// TIA Portal V19 export
FUNCTION "CollectAlarms" : Void   // FC103, LAD
TITLE = Alarm Collector Unit
// Collects alarms from the respective level and categorises the alarms into the different alarm classes. Filling the alarm DB with specific alarm messages which are defined in the comment of the defined alarm. The definition of possible alarms within a equipment is handled here.
// stored: Namespace Unit2.Em5, SetENOAutomatically false
   VAR_INPUT
      resetAlarms : Bool;
      disableAlarms : Bool;
   END_VAR
   VAR_OUTPUT
      commandsToUnit : "LUC_typeStateCommands";   // Feedback to the unit
   END_VAR
BEGIN

REGION Network 1: Reset Alarms
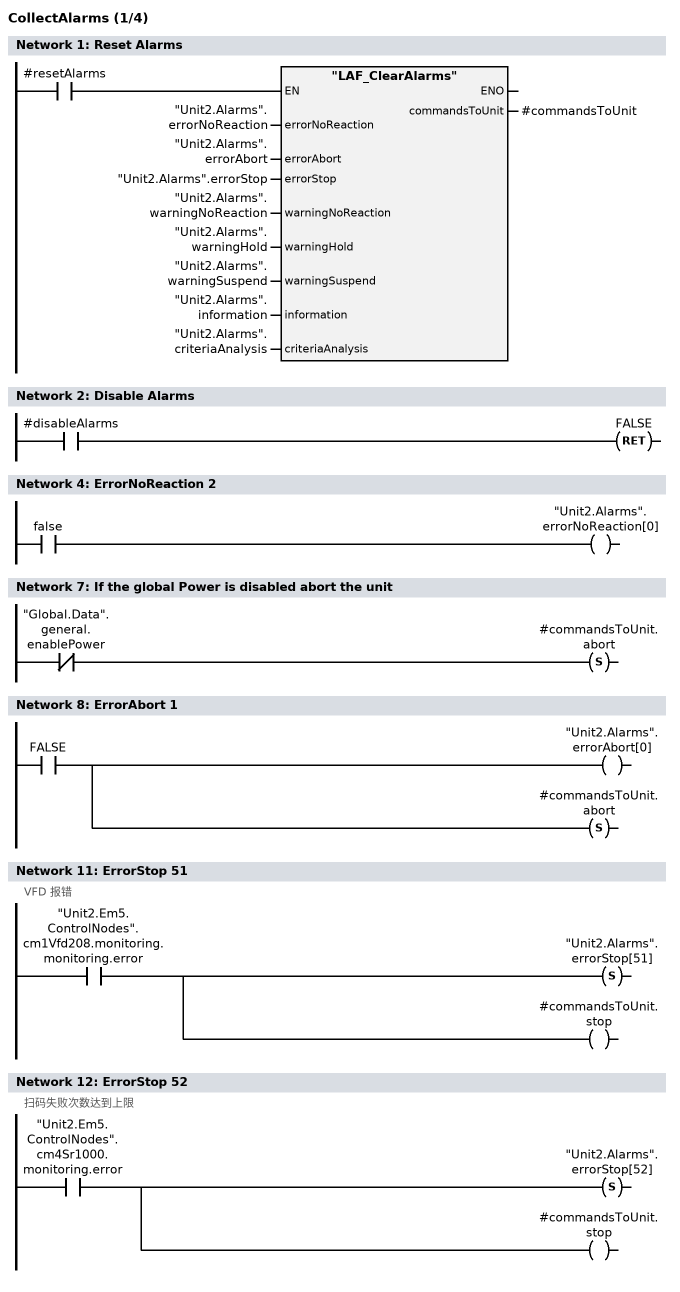
   RUNG wire#powerrail
      Contact( #resetAlarms )
      "LAF_ClearAlarms"(errorNoReaction := "Unit2.Alarms".errorNoReaction, errorAbort := "Unit2.Alarms".errorAbort, errorStop := "Unit2.Alarms".errorStop, warningNoReaction := "Unit2.Alarms".warningNoReaction, warningHold := "Unit2.Alarms".warningHold, warningSuspend := "Unit2.Alarms".warningSuspend, information := "Unit2.Alarms".information, criteriaAnalysis := "Unit2.Alarms".criteriaAnalysis, commandsToUnit => #commandsToUnit)
   END_RUNG
   // the same network as SCL:
   IF #resetAlarms THEN
       "LAF_ClearAlarms"(errorNoReaction := "Unit2.Alarms".errorNoReaction,
                         errorAbort := "Unit2.Alarms".errorAbort,
                         errorStop := "Unit2.Alarms".errorStop,
                         warningNoReaction := "Unit2.Alarms".warningNoReaction,
                         warningHold := "Unit2.Alarms".warningHold,
                         warningSuspend := "Unit2.Alarms".warningSuspend,
                         information := "Unit2.Alarms".information,
                         criteriaAnalysis := "Unit2.Alarms".criteriaAnalysis,
                         commandsToUnit => #commandsToUnit);
   END_IF;
END_REGION

REGION Network 2: Disable Alarms
   RUNG wire#powerrail
      Contact( #disableAlarms )
      ReturnCoil( FALSE )
   END_RUNG
   // the same network as SCL:
   IF #disableAlarms THEN
       ENO := FALSE;
       RETURN;
   END_IF;
END_REGION

REGION Network 3: *************** Error No Reaction ************************
END_REGION

REGION Network 4: ErrorNoReaction 2
   RUNG wire#powerrail
      Contact( false )
      Coil( "Unit2.Alarms".errorNoReaction[0] )
   END_RUNG
   // the same network as SCL:
   "Unit2.Alarms".errorNoReaction[0] := false;
END_REGION

REGION Network 6: *************** Error and Abort **************************
END_REGION

REGION Network 7: If the global Power is disabled abort the unit
   RUNG wire#powerrail
      I_Contact( "Global.Data".general.enablePower )
      S_Coil( #commandsToUnit.abort )
   END_RUNG
   // the same network as SCL:
   IF NOT "Global.Data".general.enablePower THEN #commandsToUnit.abort := TRUE; END_IF;
END_REGION

REGION Network 8: ErrorAbort 1
   RUNG wire#powerrail
      Contact( FALSE )
      wire#w1
      Coil( "Unit2.Alarms".errorAbort[0] )
   END_RUNG
   RUNG wire#w1
      S_Coil( #commandsToUnit.abort )
   END_RUNG
   // the same network as SCL:
   "Unit2.Alarms".errorAbort[0] := FALSE;
   IF FALSE THEN #commandsToUnit.abort := TRUE; END_IF;
END_REGION

REGION Network 10: *************** Error and Stop ***************************
END_REGION

REGION Network 11: ErrorStop 51
   // VFD 报错
   RUNG wire#powerrail
      Contact( "Unit2.Em5.ControlNodes".cm1Vfd208.monitoring.monitoring.error )
      wire#w1
      S_Coil( "Unit2.Alarms".errorStop[51] )
   END_RUNG
   RUNG wire#w1
      Coil( #commandsToUnit.stop )
   END_RUNG
   // the same network as SCL:
   IF "Unit2.Em5.ControlNodes".cm1Vfd208.monitoring.monitoring.error THEN
       "Unit2.Alarms".errorStop[51] := TRUE;
   END_IF;
   #commandsToUnit.stop := "Unit2.Em5.ControlNodes".cm1Vfd208.monitoring.monitoring.error;
END_REGION

REGION Network 12: ErrorStop 52
   // 扫码失败次数达到上限
   RUNG wire#powerrail
      Contact( "Unit2.Em5.ControlNodes".cm4Sr1000.monitoring.error )
      wire#w1
      S_Coil( "Unit2.Alarms".errorStop[52] )
   END_RUNG
   RUNG wire#w1
      Coil( #commandsToUnit.stop )
   END_RUNG
   // the same network as SCL:
   IF "Unit2.Em5.ControlNodes".cm4Sr1000.monitoring.error THEN "Unit2.Alarms".errorStop[52] := TRUE; END_IF;
   #commandsToUnit.stop := "Unit2.Em5.ControlNodes".cm4Sr1000.monitoring.error;
END_REGION

REGION Network 13: ErrorStop 53
   // cm2气缸报错
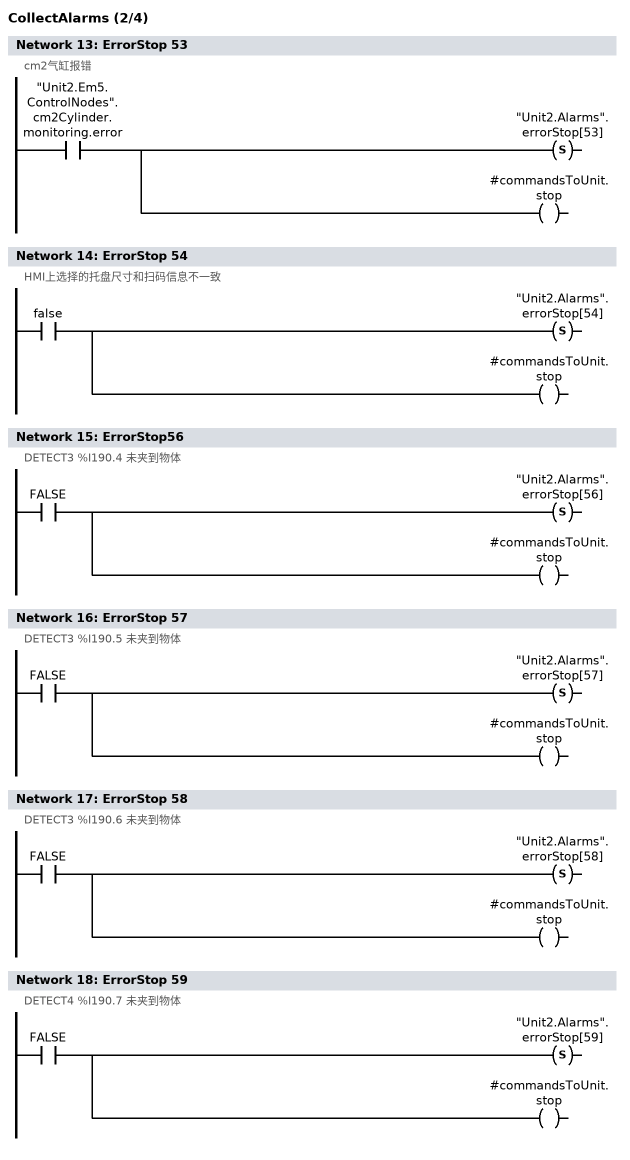
   RUNG wire#powerrail
      Contact( "Unit2.Em5.ControlNodes".cm2Cylinder.monitoring.error )
      wire#w1
      S_Coil( "Unit2.Alarms".errorStop[53] )
   END_RUNG
   RUNG wire#w1
      Coil( #commandsToUnit.stop )
   END_RUNG
   // the same network as SCL:
   IF "Unit2.Em5.ControlNodes".cm2Cylinder.monitoring.error THEN
       "Unit2.Alarms".errorStop[53] := TRUE;
   END_IF;
   #commandsToUnit.stop := "Unit2.Em5.ControlNodes".cm2Cylinder.monitoring.error;
END_REGION

REGION Network 14: ErrorStop 54
   // HMI上选择的托盘尺寸和扫码信息不一致
   RUNG wire#powerrail
      Contact( false )
      wire#w1
      S_Coil( "Unit2.Alarms".errorStop[54] )
   END_RUNG
   RUNG wire#w1
      Coil( #commandsToUnit.stop )
   END_RUNG
   // the same network as SCL:
   IF false THEN "Unit2.Alarms".errorStop[54] := TRUE; END_IF;
   #commandsToUnit.stop := false;
END_REGION

REGION Network 15: ErrorStop56
   // DETECT3 %I190.4 未夹到物体
   RUNG wire#powerrail
      Contact( FALSE )
      wire#w1
      S_Coil( "Unit2.Alarms".errorStop[56] )
   END_RUNG
   RUNG wire#w1
      Coil( #commandsToUnit.stop )
   END_RUNG
   // the same network as SCL:
   IF FALSE THEN "Unit2.Alarms".errorStop[56] := TRUE; END_IF;
   #commandsToUnit.stop := FALSE;
END_REGION

REGION Network 16: ErrorStop 57
   // DETECT3 %I190.5 未夹到物体
   RUNG wire#powerrail
      Contact( FALSE )
      wire#w1
      S_Coil( "Unit2.Alarms".errorStop[57] )
   END_RUNG
   RUNG wire#w1
      Coil( #commandsToUnit.stop )
   END_RUNG
   // the same network as SCL:
   IF FALSE THEN "Unit2.Alarms".errorStop[57] := TRUE; END_IF;
   #commandsToUnit.stop := FALSE;
END_REGION

REGION Network 17: ErrorStop 58
   // DETECT3 %I190.6 未夹到物体
   RUNG wire#powerrail
      Contact( FALSE )
      wire#w1
      S_Coil( "Unit2.Alarms".errorStop[58] )
   END_RUNG
   RUNG wire#w1
      Coil( #commandsToUnit.stop )
   END_RUNG
   // the same network as SCL:
   IF FALSE THEN "Unit2.Alarms".errorStop[58] := TRUE; END_IF;
   #commandsToUnit.stop := FALSE;
END_REGION

REGION Network 18: ErrorStop 59
   // DETECT4 %I190.7 未夹到物体
   RUNG wire#powerrail
      Contact( FALSE )
      wire#w1
      S_Coil( "Unit2.Alarms".errorStop[59] )
   END_RUNG
   RUNG wire#w1
      Coil( #commandsToUnit.stop )
   END_RUNG
   // the same network as SCL:
   IF FALSE THEN "Unit2.Alarms".errorStop[59] := TRUE; END_IF;
   #commandsToUnit.stop := FALSE;
END_REGION

REGION Network 19: ErrorStop 60
   // 条件不满足，无法恢复步骤
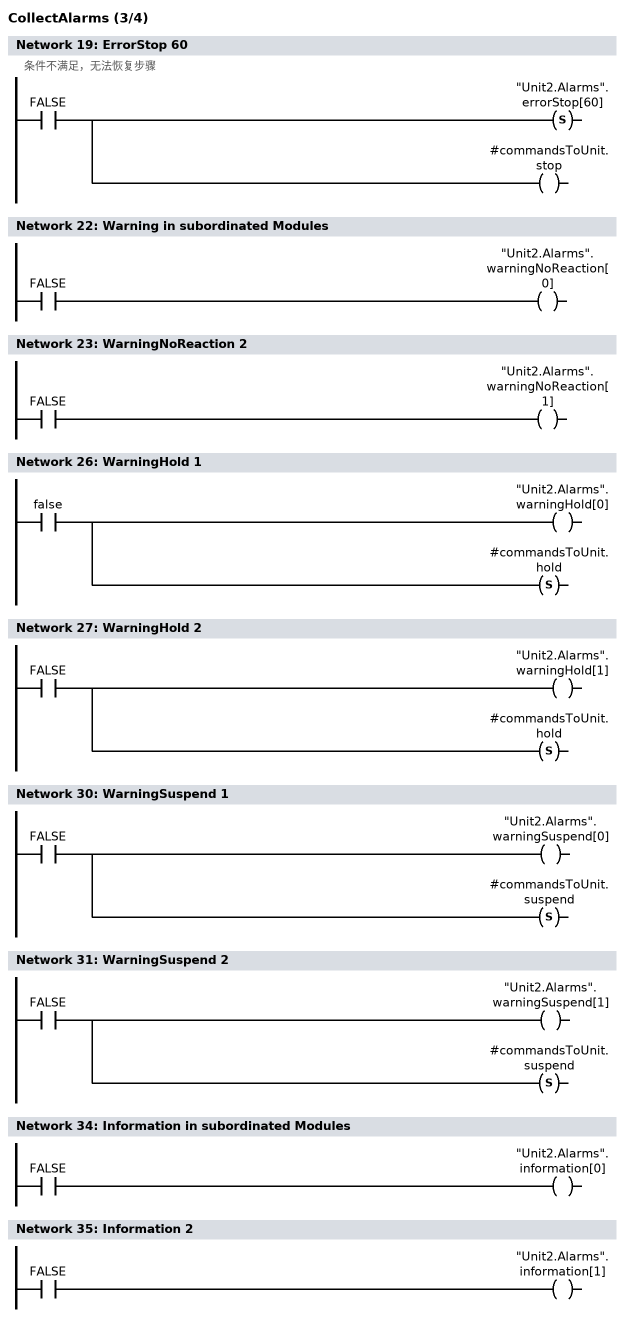
   RUNG wire#powerrail
      Contact( FALSE )
      wire#w1
      S_Coil( "Unit2.Alarms".errorStop[60] )
   END_RUNG
   RUNG wire#w1
      Coil( #commandsToUnit.stop )
   END_RUNG
   // the same network as SCL:
   IF FALSE THEN "Unit2.Alarms".errorStop[60] := TRUE; END_IF;
   #commandsToUnit.stop := FALSE;
END_REGION

REGION Network 21: *************** Warning No Reaction **********************
END_REGION

REGION Network 22: Warning in subordinated Modules
   RUNG wire#powerrail
      Contact( FALSE )
      Coil( "Unit2.Alarms".warningNoReaction[0] )
   END_RUNG
   // the same network as SCL:
   "Unit2.Alarms".warningNoReaction[0] := FALSE;
END_REGION

REGION Network 23: WarningNoReaction 2
   RUNG wire#powerrail
      Contact( FALSE )
      Coil( "Unit2.Alarms".warningNoReaction[1] )
   END_RUNG
   // the same network as SCL:
   "Unit2.Alarms".warningNoReaction[1] := FALSE;
END_REGION

REGION Network 25: *************** Warning Hold **************************
END_REGION

REGION Network 26: WarningHold 1
   RUNG wire#powerrail
      Contact( false )
      wire#w1
      Coil( "Unit2.Alarms".warningHold[0] )
   END_RUNG
   RUNG wire#w1
      S_Coil( #commandsToUnit.hold )
   END_RUNG
   // the same network as SCL:
   "Unit2.Alarms".warningHold[0] := false;
   IF false THEN #commandsToUnit.hold := TRUE; END_IF;
END_REGION

REGION Network 27: WarningHold 2
   RUNG wire#powerrail
      Contact( FALSE )
      wire#w1
      Coil( "Unit2.Alarms".warningHold[1] )
   END_RUNG
   RUNG wire#w1
      S_Coil( #commandsToUnit.hold )
   END_RUNG
   // the same network as SCL:
   "Unit2.Alarms".warningHold[1] := FALSE;
   IF FALSE THEN #commandsToUnit.hold := TRUE; END_IF;
END_REGION

REGION Network 29: *************** Warning Suspend ***********************
END_REGION

REGION Network 30: WarningSuspend 1
   RUNG wire#powerrail
      Contact( FALSE )
      wire#w1
      Coil( "Unit2.Alarms".warningSuspend[0] )
   END_RUNG
   RUNG wire#w1
      S_Coil( #commandsToUnit.suspend )
   END_RUNG
   // the same network as SCL:
   "Unit2.Alarms".warningSuspend[0] := FALSE;
   IF FALSE THEN #commandsToUnit.suspend := TRUE; END_IF;
END_REGION

REGION Network 31: WarningSuspend 2
   RUNG wire#powerrail
      Contact( FALSE )
      wire#w1
      Coil( "Unit2.Alarms".warningSuspend[1] )
   END_RUNG
   RUNG wire#w1
      S_Coil( #commandsToUnit.suspend )
   END_RUNG
   // the same network as SCL:
   "Unit2.Alarms".warningSuspend[1] := FALSE;
   IF FALSE THEN #commandsToUnit.suspend := TRUE; END_IF;
END_REGION

REGION Network 33: *************** Information *****************************
END_REGION

REGION Network 34: Information in subordinated Modules
   RUNG wire#powerrail
      Contact( FALSE )
      Coil( "Unit2.Alarms".information[0] )
   END_RUNG
   // the same network as SCL:
   "Unit2.Alarms".information[0] := FALSE;
END_REGION

REGION Network 35: Information 2
   RUNG wire#powerrail
      Contact( FALSE )
      Coil( "Unit2.Alarms".information[1] )
   END_RUNG
   // the same network as SCL:
   "Unit2.Alarms".information[1] := FALSE;
END_REGION

REGION Network 37: *************** CriteriaAnalysis **************************
END_REGION

REGION Network 38: CriteriaAnalysis 1
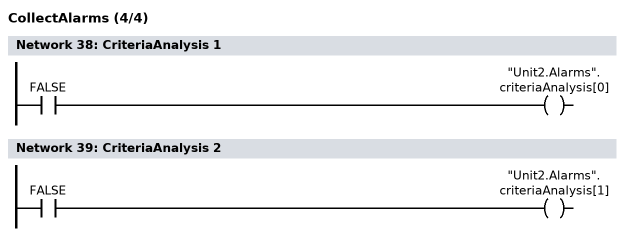
   RUNG wire#powerrail
      Contact( FALSE )
      Coil( "Unit2.Alarms".criteriaAnalysis[0] )
   END_RUNG
   // the same network as SCL:
   "Unit2.Alarms".criteriaAnalysis[0] := FALSE;
END_REGION

REGION Network 39: CriteriaAnalysis 2
   RUNG wire#powerrail
      Contact( FALSE )
      Coil( "Unit2.Alarms".criteriaAnalysis[1] )
   END_RUNG
   // the same network as SCL:
   "Unit2.Alarms".criteriaAnalysis[1] := FALSE;
END_REGION
END_FUNCTION
